FUNCTION_BLOCK xPPU_LSC
VAR_INPUT
	i_error: POINTER TO ErrorManager;
	i_process: POINTER TO ProcessManager;
	i_state: POINTER TO StateTracker;
END_VAR
VAR
	m_conveyorParams: ParameterSet;
	m_subRes: EOperationResult;
END_VAR

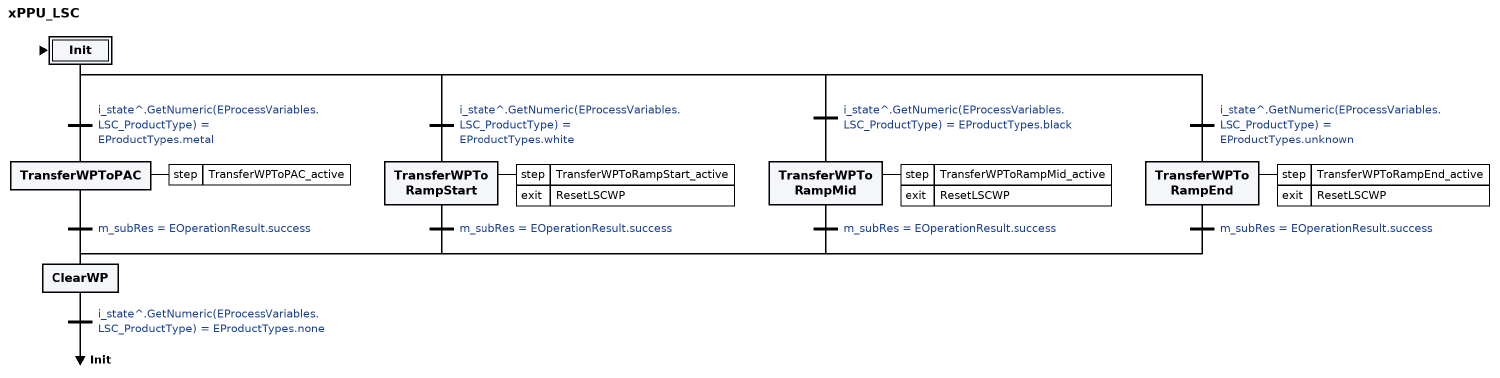
INITIAL_STEP Init:
END_STEP
TRANSITION FROM Init TO TransferWPToPAC
    := i_state^.GetNumeric(EProcessVariables.LSC_ProductType) = EProductTypes.metal;
END_TRANSITION
STEP TransferWPToPAC:
    TransferWPToPAC_active(N);  // step action
END_STEP
TRANSITION FROM TransferWPToPAC TO ClearWP
    := m_subRes = EOperationResult.success;
END_TRANSITION
TRANSITION FROM Init TO TransferWPToRampStart
    := i_state^.GetNumeric(EProcessVariables.LSC_ProductType) = EProductTypes.white;
END_TRANSITION
STEP TransferWPToRampStart:
    TransferWPToRampStart_active(N);  // step action
    ResetLSCWP(P0);  // exit action
END_STEP
TRANSITION FROM TransferWPToRampStart TO ClearWP
    := m_subRes = EOperationResult.success;
END_TRANSITION
TRANSITION FROM Init TO TransferWPToRampMid
    := i_state^.GetNumeric(EProcessVariables.LSC_ProductType) = EProductTypes.black;
END_TRANSITION
STEP TransferWPToRampMid:
    TransferWPToRampMid_active(N);  // step action
    ResetLSCWP(P0);  // exit action
END_STEP
TRANSITION FROM TransferWPToRampMid TO ClearWP
    := m_subRes = EOperationResult.success;
END_TRANSITION
TRANSITION FROM Init TO TransferWPToRampEnd
    := i_state^.GetNumeric(EProcessVariables.LSC_ProductType) = EProductTypes.unknown;
END_TRANSITION
STEP TransferWPToRampEnd:
    TransferWPToRampEnd_active(N);  // step action
    ResetLSCWP(P0);  // exit action
END_STEP
TRANSITION FROM TransferWPToRampEnd TO ClearWP
    := m_subRes = EOperationResult.success;
END_TRANSITION
STEP ClearWP:
END_STEP
TRANSITION FROM ClearWP TO Init
    := i_state^.GetNumeric(EProcessVariables.LSC_ProductType) = EProductTypes.none;
END_TRANSITION

ACTION ResetLSCWP:
i_state^.ResetProduct(EProducts.LSC_product);
END_ACTION

ACTION TransferWPToPAC_active:
m_subRes := i_process^.Execute(
	EBehaviorType.control_primitive,
	EPrimitives.LSC_TransferWorkpieceTo_PAC,
	m_conveyorParams);
END_ACTION

ACTION TransferWPToRampEnd_active:
m_subRes := i_process^.Execute(
	EBehaviorType.control_primitive,
	EPrimitives.LSC_TransferWorkpieceTo_RampEnd,
	m_conveyorParams);
END_ACTION

ACTION TransferWPToRampMid_active:
m_subRes := i_process^.Execute(
	EBehaviorType.control_primitive,
	EPrimitives.LSC_TransferWorkpieceTo_RampMid,
	m_conveyorParams);
END_ACTION

ACTION TransferWPToRampStart_active:
m_subRes := i_process^.Execute(
	EBehaviorType.control_primitive,
	EPrimitives.LSC_TransferWorkpieceTo_RampStart,
	m_conveyorParams);
END_ACTION

END_FUNCTION_BLOCK

(* stored: Version 1.1.0.1, ProductVersion 3.1.4024.4
   POU xPPU_LSC: Id {8246a5de-9303-4982-9c16-a709139cb910}, SpecialFunc None
   Action ResetLSCWP: Id {7fb1714f-6424-4786-a5e1-3c86619d5b06}
   Action TransferWPToPAC_active: Id {52233bd1-b3db-4254-98fc-82373ff14cb5}
   Action TransferWPToRampEnd_active: Id {e1536d26-ab26-4cec-8e9e-336f227510b4}
   Action TransferWPToRampMid_active: Id {4bd98ecb-0488-416f-a2ed-b9eddd1c18f1}
   Action TransferWPToRampStart_active: Id {cec12bdf-7a2b-4fd0-8f98-bc04b09d656d} *)
